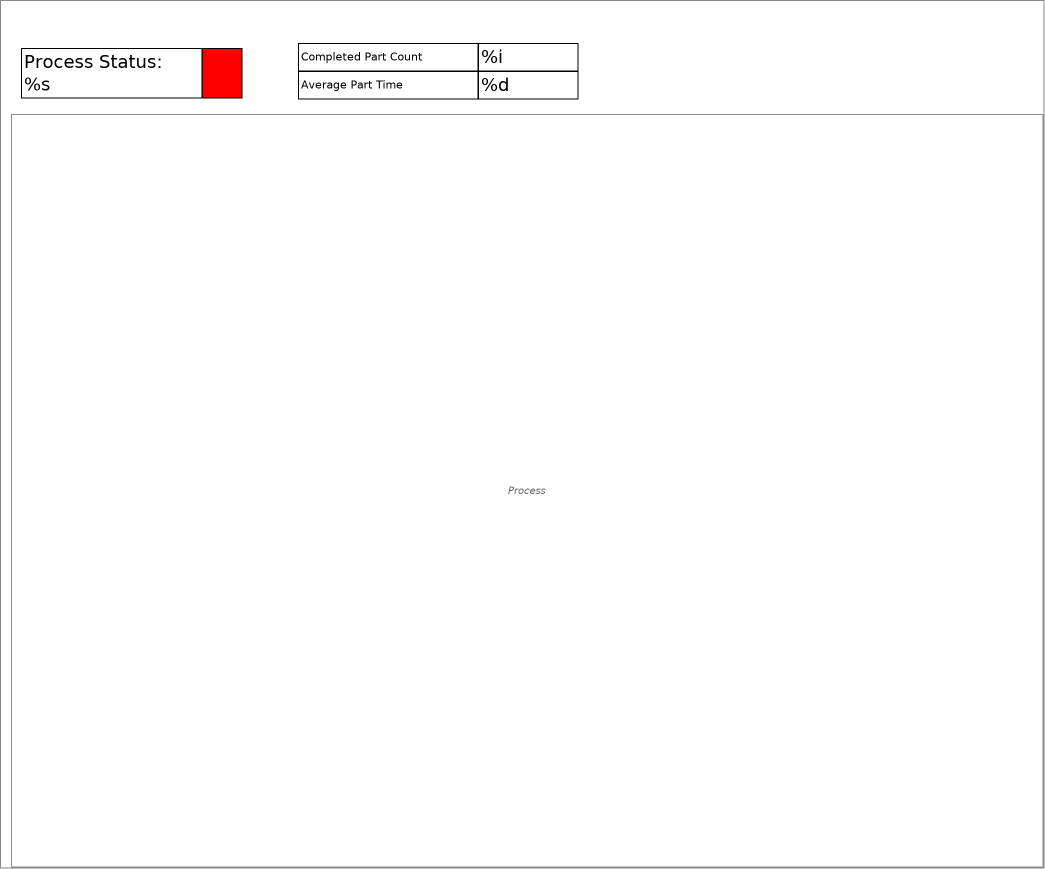
VISUALIZATION TopVisu  // 1045x869
    TabControl (11,114 1032x753)
        shows Process()
        shows PositionCheck()
        shows ForceAndTorque()
        shows Settings()
        [0]: TabTitle=System Process
        [1]: TabTitle=Position Check
        [2]: TabTitle=Force and Torqu Sensor
        [3]: TabTitle=System Settings
    Rectangle (202,48 40x50), colour toggle: MAIN.eProcessMode = E_ProcessModes.Running
    Rectangle (21,48 181x50), "Process Status: %s", text variable: MAIN.sProcessState
    Rectangle (298,43 180x28), "Completed Part Count"
    Rectangle (298,71 180x28), "Average Part Time"
    Rectangle (478,43 100x28), "%i", text variable: Global.nPartsCompleted
    Rectangle (478,71 100x28), "%d", text variable: Global.nAveragePartTime
END_VISUALIZATION

(* stored: Version 1.1.0.1, ProductVersion 3.1.4020.12
   Visu TopVisu: Id {9a9ba2a8-953c-4b64-a019-fce135ea3ba4} *)
